Fanuc KAREL source: test_shapes.kl

PROGRAM test_shapes
%NOLOCKGROUP

%include common_poses.klt
%include shapes.klt

%from systemlib.klh %import VEC
%include kunit.klh
%include shapes.klh

%class cyltst('cylinder.klc','cylinder.klh')


ROUTINE t_cyl_col : BOOLEAN
  VAR
    p : ARRAY[4] OF VECTOR
    b : ARRAY[4] OF BOOLEAN
    origin : XYZWPR
  BEGIN
    --set cylinder origin
    origin = ZEROPOS(1)
    origin.z = 270
    --create cylinder
    cyltst__new(origin, 100, 300, TRUE)

    --inside cylinder
    p[1] = VEC(30,30,290)
    --at surface of cylinder
    p[2] = VEC(60,-85,330)
    --outside cylinder
    p[3] = VEC(140,190,290)
    -- in front of cylinder
    p[4] = VEC(0,0,710)


    --test collisions
    -- radius = 100mm , start_z = 270mm, length = 300mm
    -- b1 = true
    b[1] = cyltst__point_collision(p[1])
    -- b2 = false
    b[2] = cyltst__point_collision(p[2])
    -- -- b3 = false
    b[3] = cyltst__point_collision(p[3])
    -- -- b4 = false
    b[4] = cyltst__point_collision(p[4])

    cyltst__clear

    RETURN ( kunit_assert(b[1]) AND NOT kunit_assert(b[2]) AND &
             NOT kunit_assert(b[3]) AND NOT kunit_assert(b[4]))

  END t_cyl_col

ROUTINE t_pnt2pln : BOOLEAN
  VAR
    origin : ARRAY[4] OF VECTOR
    normal : ARRAY[4] OF VECTOR
    point : ARRAY[4] OF VECTOR
    expected : ARRAY[4] OF VECTOR
    planes : ARRAY[4] OF T_PLANE
  BEGIN
    WRITE(CR,CR)
    --point above plane
    origin[1] = VEC(-2.73875,-1.91717,0.59822)
    normal[1] = VEC(2.06,1.53,1.7)
    point[1] = VEC(8.51735,-8.80025,2.73481)
    expected[1] = VEC(5.02,-11.42,-0.17)

    shapes__create_plane(origin[1], normal[1], planes[1])

    --point below plane
    origin[2] = VEC(-1.2,-3.2,0.6)
    normal[2] = VEC(-1.32,-0.43,1.7)
    point[2] = VEC(4.3,-7.1,-0.5)
    expected[2] = VEC(2.25,-7.77,2.14)

    shapes__create_plane(origin[2], normal[2], planes[2])

    --0 d
    origin[3] = VEC(0,0,0)
    normal[3] = VEC(1.58,2.83,1)
    point[3] = VEC(4.71,1.04,2.73)
    expected[3] = VEC(2.91,-2.19,1.59)

    shapes__create_plane(origin[3], normal[3], planes[3])

    --flat plane
    origin[4] = VEC(0,0,0)
    normal[4] = VEC(0,0,1)
    point[4] = VEC(-4,-2.74,-1.52)
    expected[4] = VEC(-4,-2.74,0)

    shapes__create_plane(origin[4], normal[4], planes[4])

    RETURN( kunit_eq_vrl(expected[1], shapes__project_point_on_plane(point[1], planes[1]), 0.05) AND
         kunit_eq_vrl(expected[2], shapes__project_point_on_plane(point[2], planes[2]), 0.05) AND
         kunit_eq_vrl(expected[3], shapes__project_point_on_plane(point[3], planes[3]), 0.05) AND
         kunit_eq_vrl(expected[4], shapes__project_point_on_plane(point[4], planes[4]), 0.05) )
  END t_pnt2pln

ROUTINE t_pnt2pln2 : BOOLEAN
  VAR
    setpnts1 : ARRAY[3] OF VECTOR
    setpnts2 : ARRAY[3] OF VECTOR
    actual_plane : T_PLANE
    expect_plane : T_PLANE
    b1, b2, b3, b4 : BOOLEAN
  BEGIN
    -- create plane from 3 points
    setpnts1[1] = VEC(0,0,0)
    setpnts1[2] = VEC(1,0,0)
    setpnts1[3] = VEC(0,1,0)
    actual_plane = shapes__create_plane_from_points(setpnts1[1], setpnts1[2], setpnts1[3])
    expect_plane.normal = VEC(0,0,1)
    expect_plane.origin = VEC(0,0,0)
    expect_plane.d = 0
    b1 = kunit_assert(kunit_eq_vec(expect_plane.normal, actual_plane.normal) AND kunit_eq_vec(expect_plane.origin, actual_plane.origin) AND kunit_eq_r(expect_plane.d, actual_plane.d))

    -- create plane from 3 points
    setpnts2[1] = VEC(0,0,0)
    setpnts2[2] = VEC(1,0,0)
    setpnts2[3] = VEC(0,0,1)
    actual_plane = shapes__create_plane_from_points(setpnts2[1], setpnts2[2], setpnts2[3])
    expect_plane.normal = VEC(0,-1,0)
    expect_plane.origin = VEC(0,0,0)
    expect_plane.d = 0
    b2 = kunit_assert(kunit_eq_vec(expect_plane.normal, actual_plane.normal) AND kunit_eq_vec(expect_plane.origin, actual_plane.origin) AND kunit_eq_r(expect_plane.d, actual_plane.d))

    -- create plane from 3 points
    setpnts2[1] = VEC(1,0,0)
    setpnts2[2] = VEC(0,1,0)
    setpnts2[3] = VEC(0,0,1)
    actual_plane = shapes__create_plane_from_points(setpnts2[1], setpnts2[2], setpnts2[3])
    expect_plane.normal = VEC(1,1,1)
    expect_plane.origin = VEC(1,0,0)
    expect_plane.d = -1
    b3 = kunit_assert(kunit_eq_vec(expect_plane.normal, actual_plane.normal) AND kunit_eq_vec(expect_plane.origin, actual_plane.origin) AND kunit_eq_r(expect_plane.d, actual_plane.d))

    -- create plane from 3 points
    setpnts2[1] = VEC(2,2,2)
    setpnts2[2] = VEC(-3,3,0)
    setpnts2[3] = VEC(0,0,1)
    actual_plane = shapes__create_plane_from_points(setpnts2[1], setpnts2[2], setpnts2[3])
    expect_plane.normal = VEC(-5,-1,11.99)
    expect_plane.origin = VEC(2,2,2)
    expect_plane.d = -11.99
    b4 = kunit_assert(kunit_eq_vrl(expect_plane.normal, actual_plane.normal, 0.05) AND kunit_eq_vrl(expect_plane.origin, actual_plane.origin, 0.05) AND kunit_eq_rep(expect_plane.d, actual_plane.d, 0.05))

    RETURN(b1 AND b2 AND b3 AND b4)
  END t_pnt2pln2


ROUTINE t_plnint : BOOLEAN
  VAR
    setpnts1 : ARRAY[3] OF VECTOR
    setpnts2 : ARRAY[3] OF VECTOR
    pl1, pl2 : T_PLANE
    actual_line, actual_line2 : t_LINE
    expect_line, expect_line2 : t_LINE
  BEGIN
    --plane intersection vector
    setpnts1[1] = VEC(3,0,0)
    setpnts1[2] = VEC(0,1,0)
    setpnts1[3] = VEC(0,0,1)

    setpnts2[1] = VEC(-1,0,0)
    setpnts2[2] = VEC(0,-3,0)
    setpnts2[3] = VEC(0,0,1)

    pl1 = shapes__create_plane_from_points(setpnts1[1], setpnts1[2], setpnts1[3])
    pl2 = shapes__create_plane_from_points(setpnts2[1], setpnts2[2], setpnts2[3])
    actual_line = shapes__plane_intersection_line(pl1, pl2)

    expect_line.vec = VEC(12, -12, 8)
    expect_line.point = VEC(-1.5, 1.5, 0)

    --plane intersection vector
    setpnts1[1] = VEC(-1,0,0)
    setpnts1[2] = VEC(1,0,0)
    setpnts1[3] = VEC(0,0,1)

    setpnts2[1] = VEC(0,-1,0)
    setpnts2[2] = VEC(0,1,0)
    setpnts2[3] = VEC(0,0,1)

    pl1 = shapes__create_plane_from_points(setpnts1[1], setpnts1[2], setpnts1[3])
    pl2 = shapes__create_plane_from_points(setpnts2[1], setpnts2[2], setpnts2[3])
    actual_line2 = shapes__plane_intersection_line(pl1, pl2)

    expect_line2.vec = VEC(0,0,4)
    expect_line2.point = VEC(0,0,0)

    RETURN(kunit_eq_vrl(expect_line.vec, actual_line.vec, 0.05) AND
           kunit_eq_vrl(expect_line.point, actual_line.point, 0.05) AND
           kunit_eq_vrl(expect_line2.vec, actual_line2.vec, 0.05) AND
           kunit_eq_vrl(expect_line2.point, actual_line2.point, 0.05))

  END t_plnint


BEGIN
    -- total assersions 8
    kunit_test('test straight cylinder point collision', t_cyl_col) -- assersions 4
    kunit_test('test point projection on plane', t_pnt2pln) -- assersions 4
    kunit_test('test 3 pnt plane', t_pnt2pln2) -- assersions 12
    kunit_test('test plane intersection', t_plnint) -- assersions 6

    kunit_done
END test_shapes
